// TIA Portal V16 export
// export: Created 2021-11-12T13:31:16.4325674Z, ExportSetting WithDefaults, DisplayName Totally Integrated Automation Portal, DisplayVersion V16 Update 3, DisplayName TIA Portal Version Control Interface, DisplayVersion V16 Update 2, DisplayName TIA Portal Openness, DisplayVersion V16 Update 3, DisplayName SINAMICS Startdrive Advanced, DisplayVersion V16 Update 5, DisplayName SINAMICS Startdrive G130, G150, S120, S150, SINAMICS MV, S210, DisplayVersion V16 Update 5, DisplayName SINAMICS Startdrive G110M, G120, G120C, G120D, G120P, G115D, DisplayVersion V16 Update 5, DisplayName STEP 7 Professional, DisplayVersion V16 Update 3, DisplayName STEP 7 Safety, DisplayVersion V16, DisplayName WinCC UA Professional, DisplayVersion V16 Update 3
FUNCTION_BLOCK "STD_DriveRobotABB"   // FB1226, LAD
TITLE = STD_DriveRobotABB
{ S7_Optimized_Access := 'TRUE' }
VERSION : 0.1
// Logic for robot controller - common for up to 4 robots
// stored: AutoNumber false, IsIECCheckEnabled false, IsRetainMemResEnabled false, MemoryReserve 100, SetENOAutomatically false, UDAEnableTagReadback false
   VAR_INPUT
      IS_ZoneM { ExternalAccessible := 'False'; ExternalVisible := 'False'; ExternalWritable := 'False'} : "UDT_Status_main";   // Main structure from station
      IS_ZoneS { ExternalAccessible := 'False'; ExternalVisible := 'False'; ExternalWritable := 'False'} : "UDT_Zone_Status_specific";   // Specific structure from station
      IS_CtrlSfty : "UDT_DriveRobotABB_ControllerSftyDI";   // Controller safety signals
      IS_CtrlSig : "UDT_DriveRobotABB_ControllerDI";   // Controller non-safety signals
      IB1AckSfty : Bool;   // Reset safety circuit
      IB1En : Bool;   // Enable robots operation / Zone ready to operate
      IB1Init : Bool;   // Initialize robots - start at main
      IB1StartExt : Bool;   // Start robots task - external signal
      IB1StopExt : Bool;   // Stop robots task - external signal
      IB1LimSpd : Bool;   // Set robots maximal speed to safe speed (250mm/s default)
      IB1ReqPause : Bool;   // Request to pause robots jobs
      IB1AlmSupp : Bool;   // Suppress alarms
      IB1Robot1Initialized : Bool := false;   // Robot initialization finished (set 1 if not used)
      IB1Robot2Initialized : Bool := false;   // Robot initialization finished (set 1 if not used)
      IB1Robot3Initialized : Bool := false;   // Robot initialization finished (set 1 if not used)
      IB1Robot4Initialized : Bool := false;   // Robot initialization finished (set 1 if not used)
      IT_CommTmr : Time := T#1000ms;   // Communication timeout
      IT_AckPulseTime : Time := T#200ms;   // Acknowledge pulse length
   END_VAR
   VAR_OUTPUT
      OS_Status : Struct   // Output status
         Main : "UDT_Status_main";
         Specific : "UDT_DriveRobotABB_Status_specific";
         Error : "UDT_Error01";
      END_STRUCT;
      OS_CtrlSig : "UDT_DriveRobotABB_ControllerDO";   // Output signals to controller
      OB1CtrlRun : Bool;   // Controller running in auto mode
      OB1CycleAutostop : Bool;   // Cycle signal Autostop
   END_VAR
   VAR_IN_OUT
      XS_Parameter : "UDT_DriveRobotABB_Parameter";   // Individual parameter structure
      XS_Command : "UDT_DriveRobotABB_Command";   // Individual command structure
   END_VAR
   VAR
      SS_Alarm : Struct   // Device alarms
         CommErr : Bool;   // Communication to robot lost
         EmgStop : Bool;   // Controller emergency stop
         SftyCrct : Bool;   // Controller safety circuit
         NotInAut : Bool;   // Controller is not turned into auto mode
         Res_0_4 : Bool;   // Reserve
         Res_0_5 : Bool;   // Reserve
         Res_0_6 : Bool;   // Reserve
         Res_0_7 : Bool;   // Reserve
      END_STRUCT;
      SS_Warning : Struct   // Device warnings
         SpdRdce : Bool;   // Task speed on touch panel is not 100%
         SimIO : Bool;   // At least one signal is simulated
         SMBBatt : Bool;   // SMB battery charge low
         Temp : Bool;   // CPU temperature higher than 95°C
         NoCycle : Bool;   // None robot is executing task
         Res_0_5 : Bool;   // Reserve
         Res_0_6 : Bool;   // Reserve
         Res_0_7 : Bool;   // Reserve
      END_STRUCT;
      SS_CtrlIn { S7_SetPoint := 'True'} : "UDT_DriveRobotABB_ControllerDI";   // Controller outputs
      SS_CtrlOut { S7_SetPoint := 'True'} : "UDT_DriveRobotABB_ControllerDO";   // Controller inputs
      SB1CollErr : Bool;   // Collective error from device
      SB1CollWrn : Bool;   // Collective warning from device
      SB1CtrlRdy : Bool;   // Controller ready to operation
      SB1ReqInit : Bool;   // Robots init request
      SB1ReqStart : Bool;   // Robots start request
      SB1ReqStartAtMain : Bool;   // Robots start at main request
      SB1InitPE : Bool;   // Robot init request trigger
      SB1StartAtMainPE : Bool;   // Robot init request trigger
      SB1StartExtPE : Bool;   // External start request trigger
      SB1StartTimeOut : Bool;
      ST_CommTmr { S7_SetPoint := 'True'} : TON_TIME;
      ST_RstSfty_TP { S7_SetPoint := 'True'} : TP_TIME;
      ST_RstErr_TP { S7_SetPoint := 'True'} : TP_TIME;
      ST_RstErr_TOF { S7_SetPoint := 'True'} : TOF_TIME;
      ST_ReqStartTimeOut { S7_SetPoint := 'True'} : TON_TIME;
      SS_InitSeqNr : Byte;   // Sequence Initialization
      IEC_Timer_0_Instance { S7_SetPoint := 'True'} : TON_TIME;
      ST_CycleAutostop { S7_SetPoint := 'True'} : TON_TIME;
   END_VAR
   VAR_TEMP
      TS_Status : Struct
         Main : "UDT_Status_main";
         Specific : "UDT_DriveRobotABB_Status_specific";
         Error : "UDT_Error01";
      END_STRUCT;
      TS_Parameter : "UDT_DriveRobotABB_Parameter";
      TS_Command : "UDT_DriveRobotABB_Command";
      TB1CtrlMainCond : Bool;
      TB1AckPulse : Bool;
      TB1AlmSupp : Bool;
      TB1CycleAutostop : Bool;   // Cycle signal Autostop
   END_VAR
   VAR_TEMP   // added for the SCL form of the ladder/FBD networks
      _w1 : Bool;
   END_VAR
BEGIN

REGION Network 1: Clear temporary TS_Status - Main, Specific
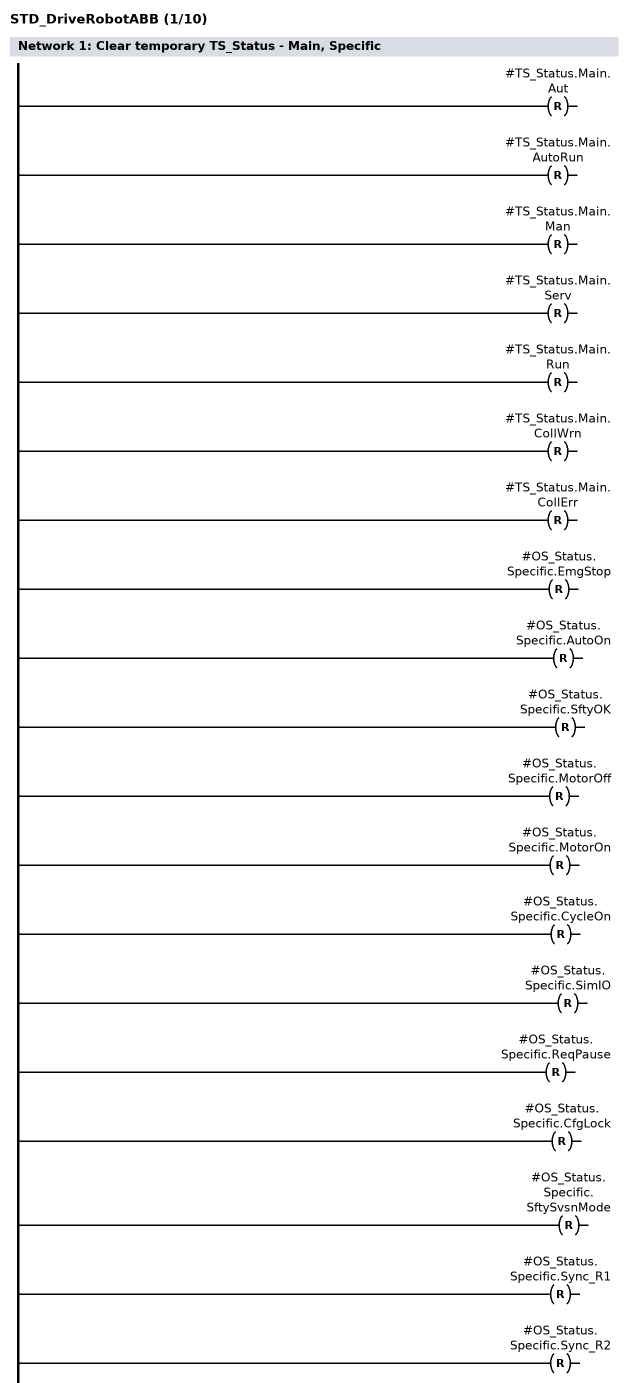
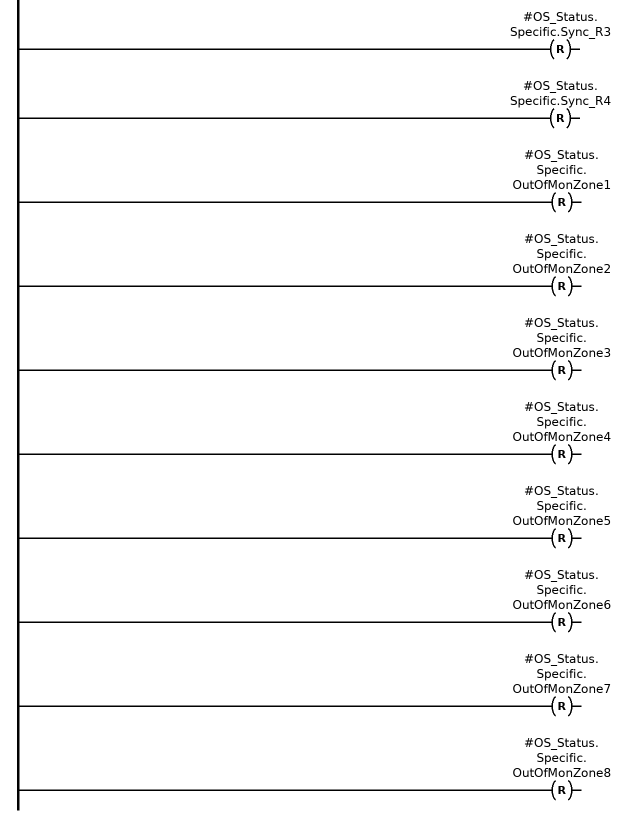
   RUNG wire#powerrail
      R_Coil( #TS_Status.Main.Aut )
   END_RUNG
   RUNG wire#powerrail
      R_Coil( #TS_Status.Main.AutoRun )
   END_RUNG
   RUNG wire#powerrail
      R_Coil( #TS_Status.Main.Man )
   END_RUNG
   RUNG wire#powerrail
      R_Coil( #TS_Status.Main.Serv )
   END_RUNG
   RUNG wire#powerrail
      R_Coil( #TS_Status.Main.Run )
   END_RUNG
   RUNG wire#powerrail
      R_Coil( #TS_Status.Main.CollWrn )
   END_RUNG
   RUNG wire#powerrail
      R_Coil( #TS_Status.Main.CollErr )
   END_RUNG
   RUNG wire#powerrail
      R_Coil( #OS_Status.Specific.EmgStop )
   END_RUNG
   RUNG wire#powerrail
      R_Coil( #OS_Status.Specific.AutoOn )
   END_RUNG
   RUNG wire#powerrail
      R_Coil( #OS_Status.Specific.SftyOK )
   END_RUNG
   RUNG wire#powerrail
      R_Coil( #OS_Status.Specific.MotorOff )
   END_RUNG
   RUNG wire#powerrail
      R_Coil( #OS_Status.Specific.MotorOn )
   END_RUNG
   RUNG wire#powerrail
      R_Coil( #OS_Status.Specific.CycleOn )
   END_RUNG
   RUNG wire#powerrail
      R_Coil( #OS_Status.Specific.SimIO )
   END_RUNG
   RUNG wire#powerrail
      R_Coil( #OS_Status.Specific.ReqPause )
   END_RUNG
   RUNG wire#powerrail
      R_Coil( #OS_Status.Specific.CfgLock )
   END_RUNG
   RUNG wire#powerrail
      R_Coil( #OS_Status.Specific.SftySvsnMode )
   END_RUNG
   RUNG wire#powerrail
      R_Coil( #OS_Status.Specific.Sync_R1 )
   END_RUNG
   RUNG wire#powerrail
      R_Coil( #OS_Status.Specific.Sync_R2 )
   END_RUNG
   RUNG wire#powerrail
      R_Coil( #OS_Status.Specific.Sync_R3 )
   END_RUNG
   RUNG wire#powerrail
      R_Coil( #OS_Status.Specific.Sync_R4 )
   END_RUNG
   RUNG wire#powerrail
      R_Coil( #OS_Status.Specific.OutOfMonZone1 )
   END_RUNG
   RUNG wire#powerrail
      R_Coil( #OS_Status.Specific.OutOfMonZone2 )
   END_RUNG
   RUNG wire#powerrail
      R_Coil( #OS_Status.Specific.OutOfMonZone3 )
   END_RUNG
   RUNG wire#powerrail
      R_Coil( #OS_Status.Specific.OutOfMonZone4 )
   END_RUNG
   RUNG wire#powerrail
      R_Coil( #OS_Status.Specific.OutOfMonZone5 )
   END_RUNG
   RUNG wire#powerrail
      R_Coil( #OS_Status.Specific.OutOfMonZone6 )
   END_RUNG
   RUNG wire#powerrail
      R_Coil( #OS_Status.Specific.OutOfMonZone7 )
   END_RUNG
   RUNG wire#powerrail
      R_Coil( #OS_Status.Specific.OutOfMonZone8 )
   END_RUNG
   // the same network as SCL:
   #TS_Status.Main.Aut := FALSE;
   #TS_Status.Main.AutoRun := FALSE;
   #TS_Status.Main.Man := FALSE;
   #TS_Status.Main.Serv := FALSE;
   #TS_Status.Main.Run := FALSE;
   #TS_Status.Main.CollWrn := FALSE;
   #TS_Status.Main.CollErr := FALSE;
   #OS_Status.Specific.EmgStop := FALSE;
   #OS_Status.Specific.AutoOn := FALSE;
   #OS_Status.Specific.SftyOK := FALSE;
   #OS_Status.Specific.MotorOff := FALSE;
   #OS_Status.Specific.MotorOn := FALSE;
   #OS_Status.Specific.CycleOn := FALSE;
   #OS_Status.Specific.SimIO := FALSE;
   #OS_Status.Specific.ReqPause := FALSE;
   #OS_Status.Specific.CfgLock := FALSE;
   #OS_Status.Specific.SftySvsnMode := FALSE;
   #OS_Status.Specific.Sync_R1 := FALSE;
   #OS_Status.Specific.Sync_R2 := FALSE;
   #OS_Status.Specific.Sync_R3 := FALSE;
   #OS_Status.Specific.Sync_R4 := FALSE;
   #OS_Status.Specific.OutOfMonZone1 := FALSE;
   #OS_Status.Specific.OutOfMonZone2 := FALSE;
   #OS_Status.Specific.OutOfMonZone3 := FALSE;
   #OS_Status.Specific.OutOfMonZone4 := FALSE;
   #OS_Status.Specific.OutOfMonZone5 := FALSE;
   #OS_Status.Specific.OutOfMonZone6 := FALSE;
   #OS_Status.Specific.OutOfMonZone7 := FALSE;
   #OS_Status.Specific.OutOfMonZone8 := FALSE;
END_REGION

REGION Network 2: Copy In/Out variables to temporary variables
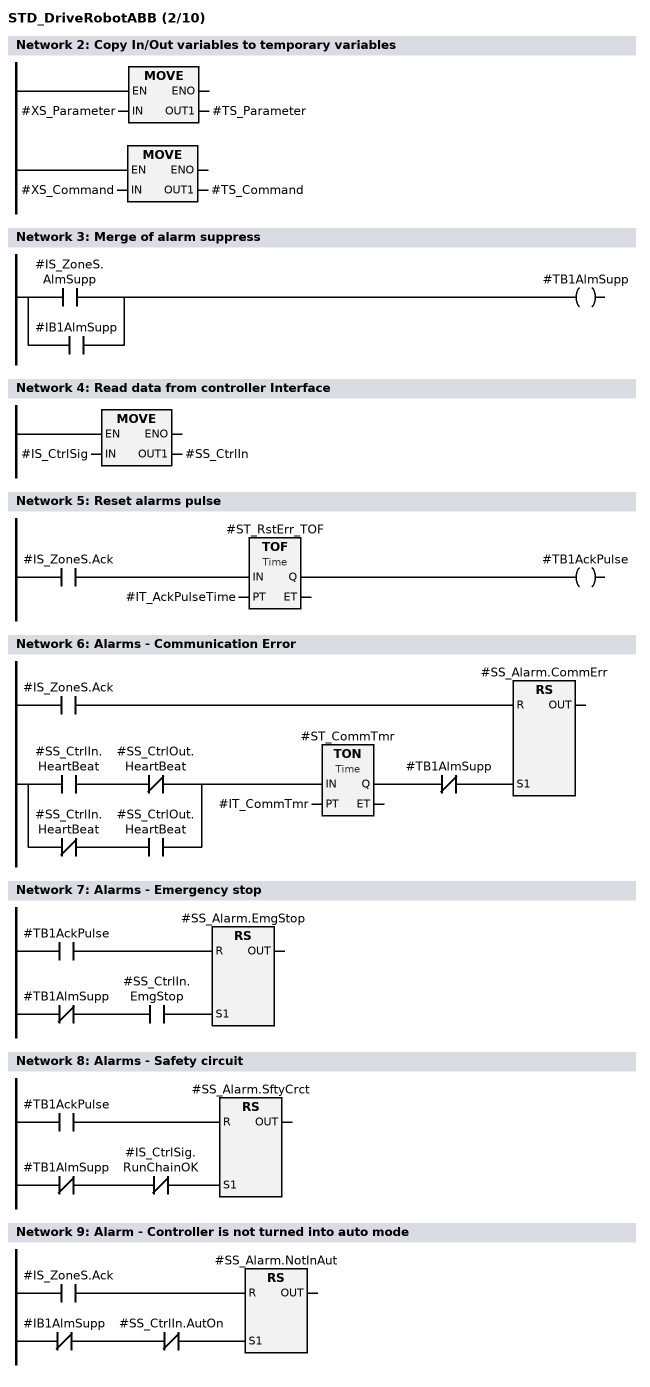
   RUNG wire#powerrail
      { S7_GenerateENO := "TRUE" } Move(in := #XS_Parameter, out1 => #TS_Parameter)
   END_RUNG
   RUNG wire#powerrail
      { S7_GenerateENO := "TRUE" } Move(in := #XS_Command, out1 => #TS_Command)
   END_RUNG
   // the same network as SCL:
   #TS_Parameter := #XS_Parameter;
   #TS_Command := #XS_Command;
END_REGION

REGION Network 3: Merge of alarm suppress
   RUNG wire#powerrail
      Contact( #IS_ZoneS.AlmSupp )
      wire#w1
      Coil( #TB1AlmSupp )
   END_RUNG
   RUNG wire#powerrail
      Contact( #IB1AlmSupp )
   END_RUNG wire#w1
   // the same network as SCL:
   #TB1AlmSupp := #IS_ZoneS.AlmSupp OR #IB1AlmSupp;
END_REGION

REGION Network 4: Read data from controller Interface
   RUNG wire#powerrail
      { S7_GenerateENO := "TRUE" } Move(in := #IS_CtrlSig, out1 => #SS_CtrlIn)
   END_RUNG
   // the same network as SCL:
   #SS_CtrlIn := #IS_CtrlSig;
END_REGION

REGION Network 5: Reset alarms pulse
   RUNG wire#powerrail
      Contact( #IS_ZoneS.Ack )
      { S7_Templates := "time_type := Time" } #ST_RstErr_TOF.TOF(pt := #IT_AckPulseTime, et =>)
      Coil( #TB1AckPulse )
   END_RUNG
   // the same network as SCL:
   #ST_RstErr_TOF(IN := #IS_ZoneS.Ack, PT := #IT_AckPulseTime);   // TOF
   #TB1AckPulse := #ST_RstErr_TOF.Q;
END_REGION

REGION Network 6: Alarms - Communication Error
   RUNG wire#powerrail
      Contact( #IS_ZoneS.Ack )
      S_RS(operand := #SS_Alarm.CommErr, s1 := wire#w2)
   END_RUNG
   RUNG wire#powerrail
      Contact( #SS_CtrlIn.HeartBeat )
      I_Contact( #SS_CtrlOut.HeartBeat )
      wire#w1
      { S7_Templates := "time_type := Time" } #ST_CommTmr.TON(pt := #IT_CommTmr, et =>)
      I_Contact( #TB1AlmSupp )
   END_RUNG wire#w2
   RUNG wire#powerrail
      I_Contact( #SS_CtrlIn.HeartBeat )
      Contact( #SS_CtrlOut.HeartBeat )
   END_RUNG wire#w1
   // the same network as SCL:
   #ST_CommTmr(IN := (#SS_CtrlIn.HeartBeat AND NOT #SS_CtrlOut.HeartBeat) OR (NOT #SS_CtrlIn.HeartBeat AND #SS_CtrlOut.HeartBeat),   // TON
               PT := #IT_CommTmr);
   IF #IS_ZoneS.Ack THEN
       #SS_Alarm.CommErr := FALSE;   // RS flip-flop
   END_IF;
   IF #ST_CommTmr.Q AND NOT #TB1AlmSupp THEN #SS_Alarm.CommErr := TRUE; END_IF;
END_REGION

REGION Network 7: Alarms - Emergency stop
   RUNG wire#powerrail
      Contact( #TB1AckPulse )
      S_RS(operand := #SS_Alarm.EmgStop, s1 := wire#w1)
   END_RUNG
   RUNG wire#powerrail
      I_Contact( #TB1AlmSupp )
      Contact( #SS_CtrlIn.EmgStop )
   END_RUNG wire#w1
   // the same network as SCL:
   IF #TB1AckPulse THEN
       #SS_Alarm.EmgStop := FALSE;   // RS flip-flop
   END_IF;
   IF NOT #TB1AlmSupp AND #SS_CtrlIn.EmgStop THEN #SS_Alarm.EmgStop := TRUE; END_IF;
END_REGION

REGION Network 8: Alarms - Safety circuit
   RUNG wire#powerrail
      Contact( #TB1AckPulse )
      S_RS(operand := #SS_Alarm.SftyCrct, s1 := wire#w1)
   END_RUNG
   RUNG wire#powerrail
      I_Contact( #TB1AlmSupp )
      I_Contact( #IS_CtrlSig.RunChainOK )
   END_RUNG wire#w1
   // the same network as SCL:
   IF #TB1AckPulse THEN
       #SS_Alarm.SftyCrct := FALSE;   // RS flip-flop
   END_IF;
   IF NOT #TB1AlmSupp AND NOT #IS_CtrlSig.RunChainOK THEN #SS_Alarm.SftyCrct := TRUE; END_IF;
END_REGION

REGION Network 9: Alarm - Controller is not turned into auto mode
   RUNG wire#powerrail
      Contact( #IS_ZoneS.Ack )
      S_RS(operand := #SS_Alarm.NotInAut, s1 := wire#w1)
   END_RUNG
   RUNG wire#powerrail
      I_Contact( #IB1AlmSupp )
      I_Contact( #SS_CtrlIn.AutOn )
   END_RUNG wire#w1
   // the same network as SCL:
   IF #IS_ZoneS.Ack THEN
       #SS_Alarm.NotInAut := FALSE;   // RS flip-flop
   END_IF;
   IF NOT #IB1AlmSupp AND NOT #SS_CtrlIn.AutOn THEN #SS_Alarm.NotInAut := TRUE; END_IF;
END_REGION

REGION Network 10: Warning - Simulated IO
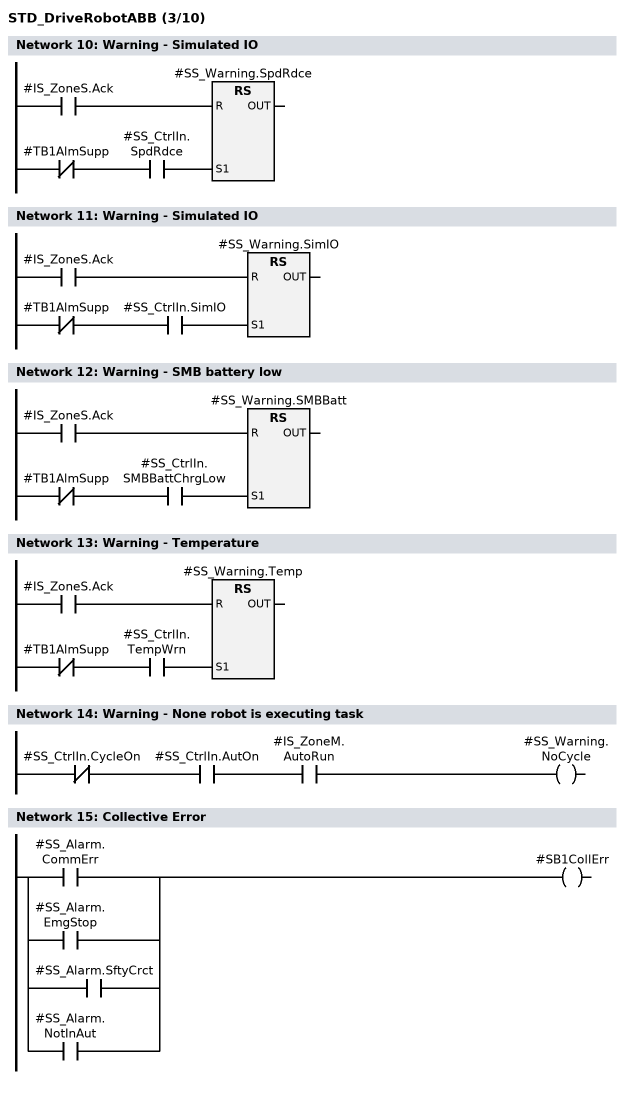
   RUNG wire#powerrail
      Contact( #IS_ZoneS.Ack )
      S_RS(operand := #SS_Warning.SpdRdce, s1 := wire#w1)
   END_RUNG
   RUNG wire#powerrail
      I_Contact( #TB1AlmSupp )
      Contact( #SS_CtrlIn.SpdRdce )
   END_RUNG wire#w1
   // the same network as SCL:
   IF #IS_ZoneS.Ack THEN
       #SS_Warning.SpdRdce := FALSE;   // RS flip-flop
   END_IF;
   IF NOT #TB1AlmSupp AND #SS_CtrlIn.SpdRdce THEN #SS_Warning.SpdRdce := TRUE; END_IF;
END_REGION

REGION Network 11: Warning - Simulated IO
   RUNG wire#powerrail
      Contact( #IS_ZoneS.Ack )
      S_RS(operand := #SS_Warning.SimIO, s1 := wire#w1)
   END_RUNG
   RUNG wire#powerrail
      I_Contact( #TB1AlmSupp )
      Contact( #SS_CtrlIn.SimIO )
   END_RUNG wire#w1
   // the same network as SCL:
   IF #IS_ZoneS.Ack THEN
       #SS_Warning.SimIO := FALSE;   // RS flip-flop
   END_IF;
   IF NOT #TB1AlmSupp AND #SS_CtrlIn.SimIO THEN #SS_Warning.SimIO := TRUE; END_IF;
END_REGION

REGION Network 12: Warning - SMB battery low
   RUNG wire#powerrail
      Contact( #IS_ZoneS.Ack )
      S_RS(operand := #SS_Warning.SMBBatt, s1 := wire#w1)
   END_RUNG
   RUNG wire#powerrail
      I_Contact( #TB1AlmSupp )
      Contact( #SS_CtrlIn.SMBBattChrgLow )
   END_RUNG wire#w1
   // the same network as SCL:
   IF #IS_ZoneS.Ack THEN
       #SS_Warning.SMBBatt := FALSE;   // RS flip-flop
   END_IF;
   IF NOT #TB1AlmSupp AND #SS_CtrlIn.SMBBattChrgLow THEN #SS_Warning.SMBBatt := TRUE; END_IF;
END_REGION

REGION Network 13: Warning - Temperature
   RUNG wire#powerrail
      Contact( #IS_ZoneS.Ack )
      S_RS(operand := #SS_Warning.Temp, s1 := wire#w1)
   END_RUNG
   RUNG wire#powerrail
      I_Contact( #TB1AlmSupp )
      Contact( #SS_CtrlIn.TempWrn )
   END_RUNG wire#w1
   // the same network as SCL:
   IF #IS_ZoneS.Ack THEN
       #SS_Warning.Temp := FALSE;   // RS flip-flop
   END_IF;
   IF NOT #TB1AlmSupp AND #SS_CtrlIn.TempWrn THEN #SS_Warning.Temp := TRUE; END_IF;
END_REGION

REGION Network 14: Warning - None robot is executing task
   RUNG wire#powerrail
      I_Contact( #SS_CtrlIn.CycleOn )
      Contact( #SS_CtrlIn.AutOn )
      Contact( #IS_ZoneM.AutoRun )
      Coil( #SS_Warning.NoCycle )
   END_RUNG
   // the same network as SCL:
   #SS_Warning.NoCycle := NOT #SS_CtrlIn.CycleOn AND #SS_CtrlIn.AutOn AND #IS_ZoneM.AutoRun;
END_REGION

REGION Network 15: Collective Error
   RUNG wire#powerrail
      Contact( #SS_Alarm.CommErr )
      wire#w1
      Coil( #SB1CollErr )
   END_RUNG
   RUNG wire#powerrail
      Contact( #SS_Alarm.EmgStop )
   END_RUNG wire#w1
   RUNG wire#powerrail
      Contact( #SS_Alarm.SftyCrct )
   END_RUNG wire#w1
   RUNG wire#powerrail
      Contact( #SS_Alarm.NotInAut )
   END_RUNG wire#w1
   // the same network as SCL:
   #SB1CollErr := #SS_Alarm.CommErr OR #SS_Alarm.EmgStop OR #SS_Alarm.SftyCrct OR #SS_Alarm.NotInAut;
END_REGION

REGION Network 16: Collective Warning
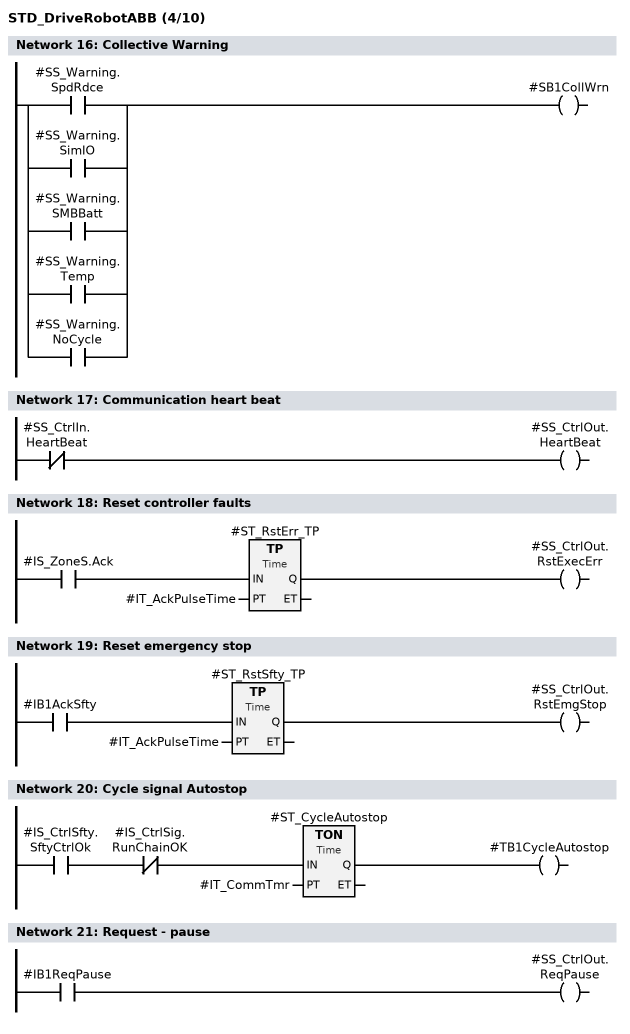
   RUNG wire#powerrail
      Contact( #SS_Warning.SpdRdce )
      wire#w1
      Coil( #SB1CollWrn )
   END_RUNG
   RUNG wire#powerrail
      Contact( #SS_Warning.SimIO )
   END_RUNG wire#w1
   RUNG wire#powerrail
      Contact( #SS_Warning.SMBBatt )
   END_RUNG wire#w1
   RUNG wire#powerrail
      Contact( #SS_Warning.Temp )
   END_RUNG wire#w1
   RUNG wire#powerrail
      Contact( #SS_Warning.NoCycle )
   END_RUNG wire#w1
   // the same network as SCL:
   #SB1CollWrn := #SS_Warning.SpdRdce OR #SS_Warning.SimIO OR #SS_Warning.SMBBatt OR #SS_Warning.Temp OR #SS_Warning.NoCycle;
END_REGION

REGION Network 17: Communication heart beat
   RUNG wire#powerrail
      I_Contact( #SS_CtrlIn.HeartBeat )
      Coil( #SS_CtrlOut.HeartBeat )
   END_RUNG
   // the same network as SCL:
   #SS_CtrlOut.HeartBeat := NOT #SS_CtrlIn.HeartBeat;
END_REGION

REGION Network 18: Reset controller faults
   RUNG wire#powerrail
      Contact( #IS_ZoneS.Ack )
      { S7_Templates := "time_type := Time" } #ST_RstErr_TP.TP(pt := #IT_AckPulseTime, et =>)
      Coil( #SS_CtrlOut.RstExecErr )
   END_RUNG
   // the same network as SCL:
   #ST_RstErr_TP(IN := #IS_ZoneS.Ack, PT := #IT_AckPulseTime);   // TP
   #SS_CtrlOut.RstExecErr := #ST_RstErr_TP.Q;
END_REGION

REGION Network 19: Reset emergency stop
   RUNG wire#powerrail
      Contact( #IB1AckSfty )
      { S7_Templates := "time_type := Time" } #ST_RstSfty_TP.TP(pt := #IT_AckPulseTime, et =>)
      Coil( #SS_CtrlOut.RstEmgStop )
   END_RUNG
   // the same network as SCL:
   #ST_RstSfty_TP(IN := #IB1AckSfty, PT := #IT_AckPulseTime);   // TP
   #SS_CtrlOut.RstEmgStop := #ST_RstSfty_TP.Q;
END_REGION

REGION Network 20: Cycle signal Autostop
   RUNG wire#powerrail
      Contact( #IS_CtrlSfty.SftyCtrlOk )
      I_Contact( #IS_CtrlSig.RunChainOK )
      { S7_Templates := "time_type := Time" } #ST_CycleAutostop.TON(pt := #IT_CommTmr, et =>)
      Coil( #TB1CycleAutostop )
   END_RUNG
   // the same network as SCL:
   #ST_CycleAutostop(IN := #IS_CtrlSfty.SftyCtrlOk AND NOT #IS_CtrlSig.RunChainOK, PT := #IT_CommTmr);   // TON
   #TB1CycleAutostop := #ST_CycleAutostop.Q;
END_REGION

REGION Network 21: Request - pause
   RUNG wire#powerrail
      Contact( #IB1ReqPause )
      Coil( #SS_CtrlOut.ReqPause )
   END_RUNG
   // the same network as SCL:
   #SS_CtrlOut.ReqPause := #IB1ReqPause;
END_REGION

REGION Network 22: Request - Start
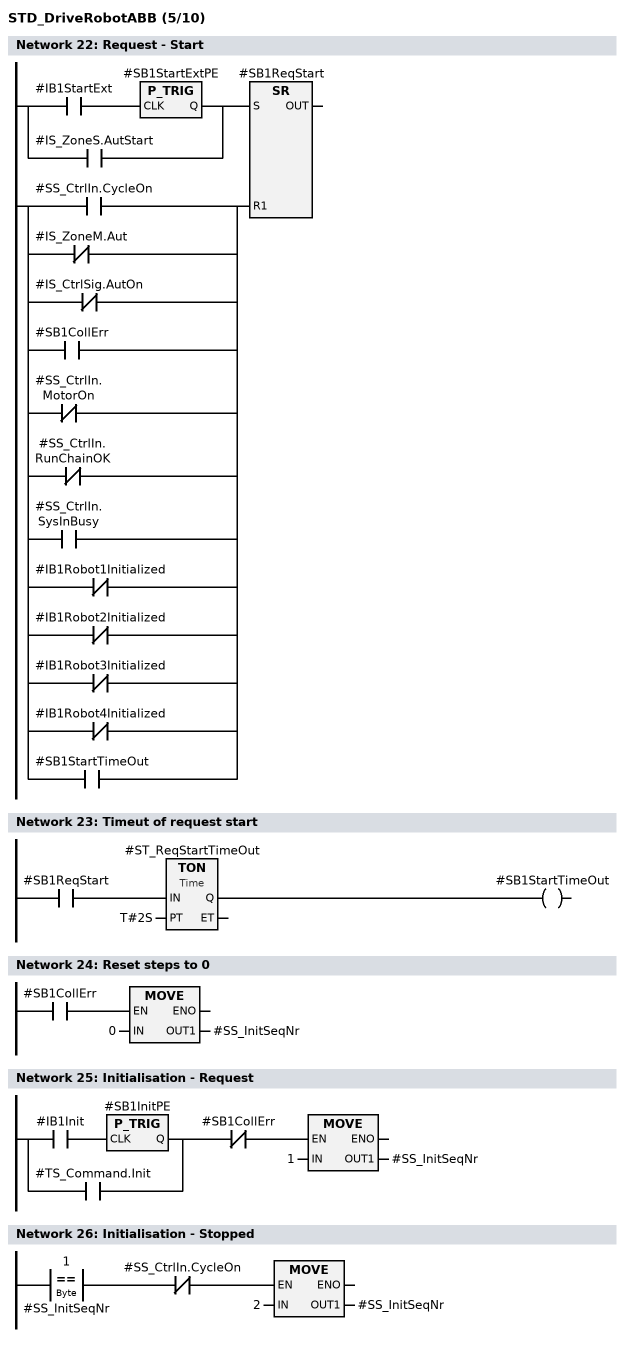
   RUNG wire#powerrail
      Contact( #IB1StartExt )
      P_Trig( #SB1StartExtPE )
      wire#w1
      S_SR(operand := #SB1ReqStart, r1 := wire#w2)
   END_RUNG
   RUNG wire#powerrail
      Contact( #IS_ZoneS.AutStart )
   END_RUNG wire#w1
   RUNG wire#powerrail
      Contact( #SS_CtrlIn.CycleOn )
   END_RUNG wire#w2
   RUNG wire#powerrail
      I_Contact( #IS_ZoneM.Aut )
   END_RUNG wire#w2
   RUNG wire#powerrail
      I_Contact( #IS_CtrlSig.AutOn )
   END_RUNG wire#w2
   RUNG wire#powerrail
      Contact( #SB1CollErr )
   END_RUNG wire#w2
   RUNG wire#powerrail
      I_Contact( #SS_CtrlIn.MotorOn )
   END_RUNG wire#w2
   RUNG wire#powerrail
      I_Contact( #SS_CtrlIn.RunChainOK )
   END_RUNG wire#w2
   RUNG wire#powerrail
      Contact( #SS_CtrlIn.SysInBusy )
   END_RUNG wire#w2
   RUNG wire#powerrail
      I_Contact( #IB1Robot1Initialized )
   END_RUNG wire#w2
   RUNG wire#powerrail
      I_Contact( #IB1Robot2Initialized )
   END_RUNG wire#w2
   RUNG wire#powerrail
      I_Contact( #IB1Robot3Initialized )
   END_RUNG wire#w2
   RUNG wire#powerrail
      I_Contact( #IB1Robot4Initialized )
   END_RUNG wire#w2
   RUNG wire#powerrail
      Contact( #SB1StartTimeOut )
   END_RUNG wire#w2
   // the same network as SCL:
   #_w1 := #IB1StartExt AND NOT #SB1StartExtPE;   // rising edge
   #SB1StartExtPE := #IB1StartExt;
   IF #_w1 OR #IS_ZoneS.AutStart THEN
       #SB1ReqStart := TRUE;   // SR flip-flop
   END_IF;
   IF #SS_CtrlIn.CycleOn OR NOT #IS_ZoneM.Aut OR NOT #IS_CtrlSig.AutOn OR #SB1CollErr OR NOT #SS_CtrlIn.MotorOn OR NOT #SS_CtrlIn.RunChainOK OR #SS_CtrlIn.SysInBusy OR NOT #IB1Robot1Initialized OR NOT #IB1Robot2Initialized OR NOT #IB1Robot3Initialized OR NOT #IB1Robot4Initialized OR #SB1StartTimeOut THEN
       #SB1ReqStart := FALSE;
   END_IF;
END_REGION

REGION Network 23: Timeut of request start
   RUNG wire#powerrail
      Contact( #SB1ReqStart )
      { S7_Templates := "time_type := Time" } #ST_ReqStartTimeOut.TON(pt := T#2S, et =>)
      Coil( #SB1StartTimeOut )
   END_RUNG
   // the same network as SCL:
   #ST_ReqStartTimeOut(IN := #SB1ReqStart, PT := T#2S);   // TON
   #SB1StartTimeOut := #ST_ReqStartTimeOut.Q;
END_REGION

REGION Network 24: Reset steps to 0
   RUNG wire#powerrail
      Contact( #SB1CollErr )
      Move(in := 0, out1 => #SS_InitSeqNr)
   END_RUNG
   // the same network as SCL:
   IF #SB1CollErr THEN #SS_InitSeqNr := 0; END_IF;
END_REGION

REGION Network 25: Initialisation - Request
   RUNG wire#powerrail
      Contact( #IB1Init )
      P_Trig( #SB1InitPE )
      wire#w1
      I_Contact( #SB1CollErr )
      Move(in := 1, out1 => #SS_InitSeqNr)
   END_RUNG
   RUNG wire#powerrail
      Contact( #TS_Command.Init )
   END_RUNG wire#w1
   // the same network as SCL:
   #_w1 := #IB1Init AND NOT #SB1InitPE;   // rising edge
   #SB1InitPE := #IB1Init;
   IF (#_w1 OR #TS_Command.Init) AND NOT #SB1CollErr THEN #SS_InitSeqNr := 1; END_IF;
END_REGION

REGION Network 26: Initialisation - Stopped
   RUNG wire#powerrail
      { S7_Templates := "SrcType := Byte" } EQ_Contact(in1 := 1, in2 := #SS_InitSeqNr)
      I_Contact( #SS_CtrlIn.CycleOn )
      Move(in := 2, out1 => #SS_InitSeqNr)
   END_RUNG
   // the same network as SCL:
   IF (1 = #SS_InitSeqNr) AND NOT #SS_CtrlIn.CycleOn THEN #SS_InitSeqNr := 2; END_IF;
END_REGION

REGION Network 27: Initialization - Started
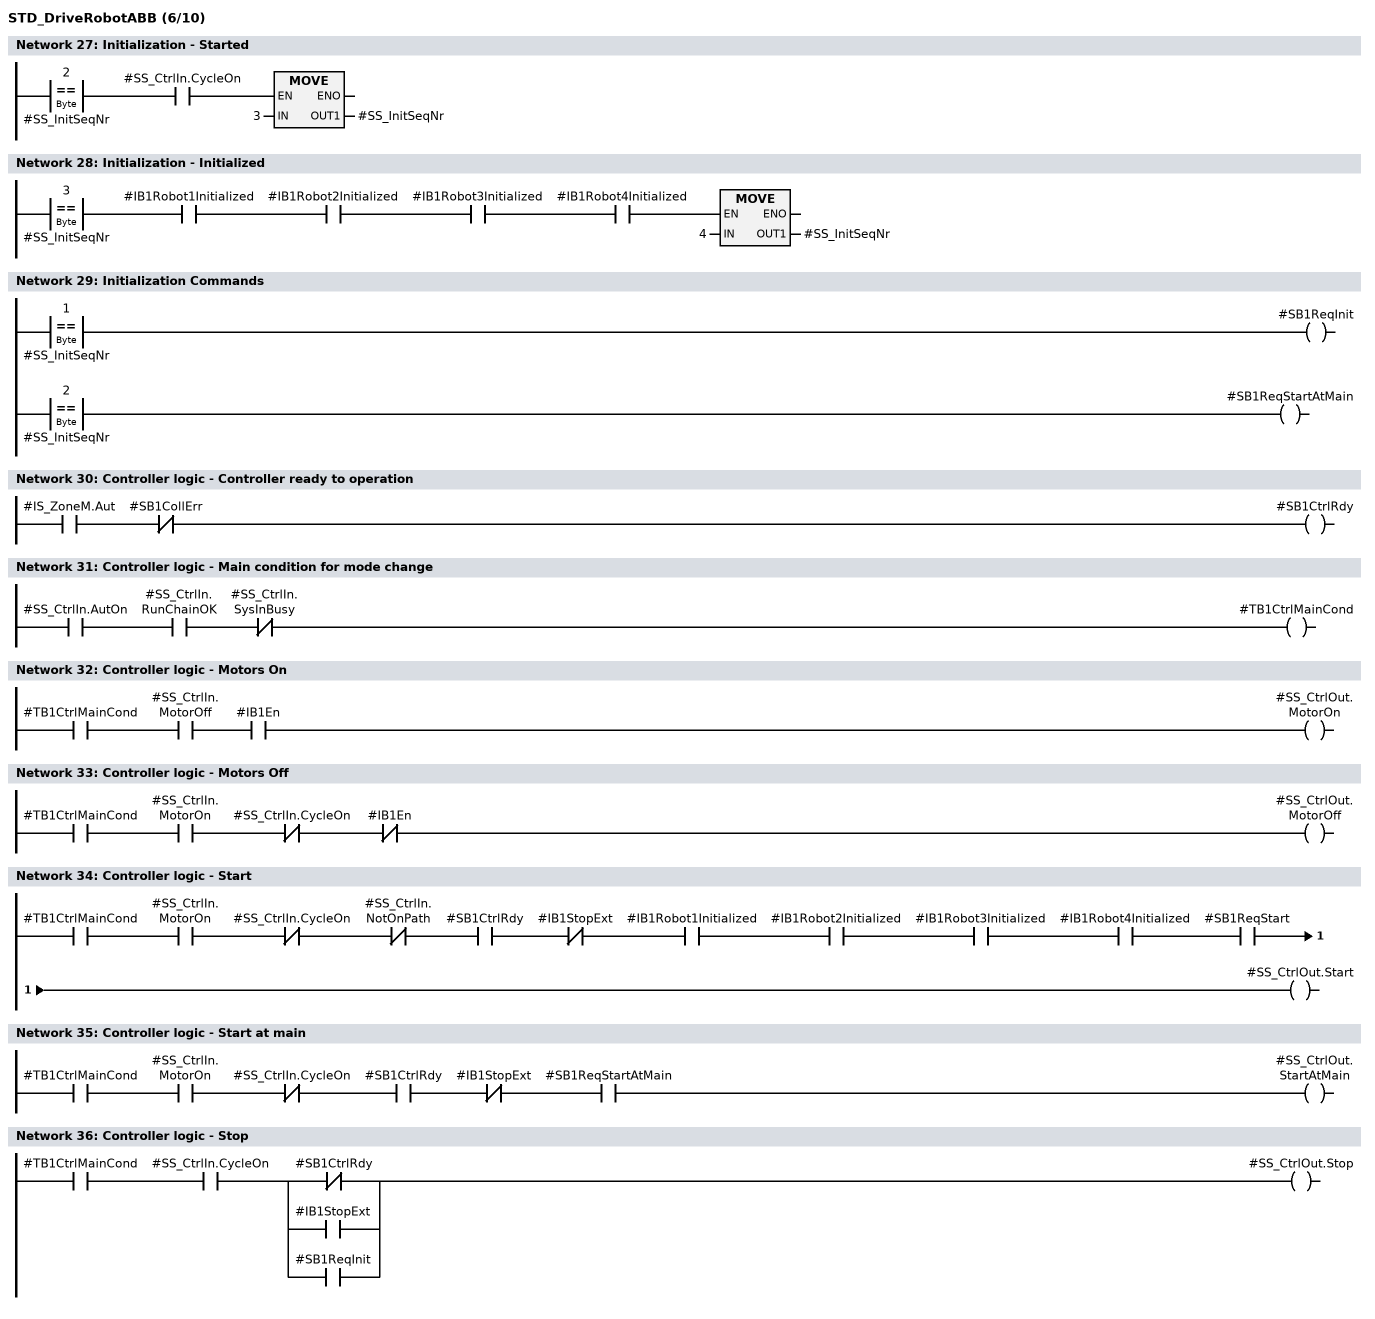
   RUNG wire#powerrail
      { S7_Templates := "SrcType := Byte" } EQ_Contact(in1 := 2, in2 := #SS_InitSeqNr)
      Contact( #SS_CtrlIn.CycleOn )
      Move(in := 3, out1 => #SS_InitSeqNr)
   END_RUNG
   // the same network as SCL:
   IF (2 = #SS_InitSeqNr) AND #SS_CtrlIn.CycleOn THEN #SS_InitSeqNr := 3; END_IF;
END_REGION

REGION Network 28: Initialization - Initialized
   RUNG wire#powerrail
      { S7_Templates := "SrcType := Byte" } EQ_Contact(in1 := 3, in2 := #SS_InitSeqNr)
      Contact( #IB1Robot1Initialized )
      Contact( #IB1Robot2Initialized )
      Contact( #IB1Robot3Initialized )
      Contact( #IB1Robot4Initialized )
      { S7_GenerateENO := "TRUE" } Move(in := 4, out1 => #SS_InitSeqNr)
   END_RUNG
   // the same network as SCL:
   IF (3 = #SS_InitSeqNr) AND #IB1Robot1Initialized AND #IB1Robot2Initialized AND #IB1Robot3Initialized AND #IB1Robot4Initialized THEN
       #SS_InitSeqNr := 4;
   END_IF;
END_REGION

REGION Network 29: Initialization Commands
   RUNG wire#powerrail
      { S7_Templates := "SrcType := Byte" } EQ_Contact(in1 := 1, in2 := #SS_InitSeqNr)
      Coil( #SB1ReqInit )
   END_RUNG
   RUNG wire#powerrail
      { S7_Templates := "SrcType := Byte" } EQ_Contact(in1 := 2, in2 := #SS_InitSeqNr)
      Coil( #SB1ReqStartAtMain )
   END_RUNG
   // the same network as SCL:
   #SB1ReqInit := 1 = #SS_InitSeqNr;
   #SB1ReqStartAtMain := 2 = #SS_InitSeqNr;
END_REGION

REGION Network 30: Controller logic - Controller ready to operation
   RUNG wire#powerrail
      Contact( #IS_ZoneM.Aut )
      I_Contact( #SB1CollErr )
      Coil( #SB1CtrlRdy )
   END_RUNG
   // the same network as SCL:
   #SB1CtrlRdy := #IS_ZoneM.Aut AND NOT #SB1CollErr;
END_REGION

REGION Network 31: Controller logic - Main condition for mode change
   RUNG wire#powerrail
      Contact( #SS_CtrlIn.AutOn )
      Contact( #SS_CtrlIn.RunChainOK )
      I_Contact( #SS_CtrlIn.SysInBusy )
      Coil( #TB1CtrlMainCond )
   END_RUNG
   // the same network as SCL:
   #TB1CtrlMainCond := #SS_CtrlIn.AutOn AND #SS_CtrlIn.RunChainOK AND NOT #SS_CtrlIn.SysInBusy;
END_REGION

REGION Network 32: Controller logic - Motors On
   RUNG wire#powerrail
      Contact( #TB1CtrlMainCond )
      Contact( #SS_CtrlIn.MotorOff )
      Contact( #IB1En )
      Coil( #SS_CtrlOut.MotorOn )
   END_RUNG
   // the same network as SCL:
   #SS_CtrlOut.MotorOn := #TB1CtrlMainCond AND #SS_CtrlIn.MotorOff AND #IB1En;
END_REGION

REGION Network 33: Controller logic - Motors Off
   RUNG wire#powerrail
      Contact( #TB1CtrlMainCond )
      Contact( #SS_CtrlIn.MotorOn )
      I_Contact( #SS_CtrlIn.CycleOn )
      I_Contact( #IB1En )
      Coil( #SS_CtrlOut.MotorOff )
   END_RUNG
   // the same network as SCL:
   #SS_CtrlOut.MotorOff := #TB1CtrlMainCond AND #SS_CtrlIn.MotorOn AND NOT #SS_CtrlIn.CycleOn AND NOT #IB1En;
END_REGION

REGION Network 34: Controller logic - Start
   RUNG wire#powerrail
      Contact( #TB1CtrlMainCond )
      Contact( #SS_CtrlIn.MotorOn )
      I_Contact( #SS_CtrlIn.CycleOn )
      I_Contact( #SS_CtrlIn.NotOnPath )
      Contact( #SB1CtrlRdy )
      I_Contact( #IB1StopExt )
      Contact( #IB1Robot1Initialized )
      Contact( #IB1Robot2Initialized )
      Contact( #IB1Robot3Initialized )
      Contact( #IB1Robot4Initialized )
      Contact( #SB1ReqStart )
      Coil( #SS_CtrlOut.Start )
   END_RUNG
   // the same network as SCL:
   #SS_CtrlOut.Start := #TB1CtrlMainCond AND #SS_CtrlIn.MotorOn AND NOT #SS_CtrlIn.CycleOn AND NOT #SS_CtrlIn.NotOnPath AND #SB1CtrlRdy AND NOT #IB1StopExt AND #IB1Robot1Initialized AND #IB1Robot2Initialized AND #IB1Robot3Initialized AND #IB1Robot4Initialized AND #SB1ReqStart;
END_REGION

REGION Network 35: Controller logic - Start at main
   RUNG wire#powerrail
      Contact( #TB1CtrlMainCond )
      Contact( #SS_CtrlIn.MotorOn )
      I_Contact( #SS_CtrlIn.CycleOn )
      Contact( #SB1CtrlRdy )
      I_Contact( #IB1StopExt )
      Contact( #SB1ReqStartAtMain )
      Coil( #SS_CtrlOut.StartAtMain )
   END_RUNG
   // the same network as SCL:
   #SS_CtrlOut.StartAtMain := #TB1CtrlMainCond AND #SS_CtrlIn.MotorOn AND NOT #SS_CtrlIn.CycleOn AND #SB1CtrlRdy AND NOT #IB1StopExt AND #SB1ReqStartAtMain;
END_REGION

REGION Network 36: Controller logic - Stop
   RUNG wire#powerrail
      Contact( #TB1CtrlMainCond )
      Contact( #SS_CtrlIn.CycleOn )
      wire#w1
      I_Contact( #SB1CtrlRdy )
      wire#w2
      Coil( #SS_CtrlOut.Stop )
   END_RUNG
   RUNG wire#w1
      Contact( #IB1StopExt )
   END_RUNG wire#w2
   RUNG wire#w1
      Contact( #SB1ReqInit )
   END_RUNG wire#w2
   // the same network as SCL:
   #SS_CtrlOut.Stop := #TB1CtrlMainCond AND #SS_CtrlIn.CycleOn AND (NOT #SB1CtrlRdy OR #IB1StopExt OR #SB1ReqInit);
END_REGION

REGION Network 37: Filling the Main status
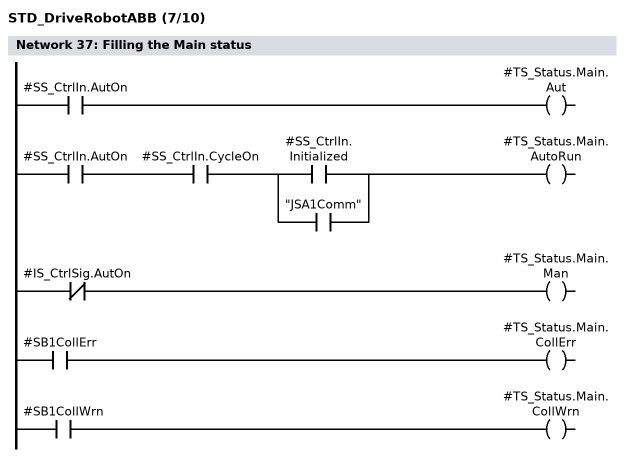
   RUNG wire#powerrail
      Contact( #SS_CtrlIn.AutOn )
      Coil( #TS_Status.Main.Aut )
   END_RUNG
   RUNG wire#powerrail
      Contact( #SS_CtrlIn.AutOn )
      Contact( #SS_CtrlIn.CycleOn )
      wire#w1
      Contact( #SS_CtrlIn.Initialized )
      wire#w2
      Coil( #TS_Status.Main.AutoRun )
   END_RUNG
   RUNG wire#w1
      Contact( "JSA1Comm" )
   END_RUNG wire#w2
   RUNG wire#powerrail
      I_Contact( #IS_CtrlSig.AutOn )
      Coil( #TS_Status.Main.Man )
   END_RUNG
   RUNG wire#powerrail
      Contact( #SB1CollErr )
      Coil( #TS_Status.Main.CollErr )
   END_RUNG
   RUNG wire#powerrail
      Contact( #SB1CollWrn )
      Coil( #TS_Status.Main.CollWrn )
   END_RUNG
   // the same network as SCL:
   #TS_Status.Main.Aut := #SS_CtrlIn.AutOn;
   #TS_Status.Main.AutoRun := #SS_CtrlIn.AutOn AND #SS_CtrlIn.CycleOn AND (#SS_CtrlIn.Initialized OR "JSA1Comm");
   #TS_Status.Main.Man := NOT #IS_CtrlSig.AutOn;
   #TS_Status.Main.CollErr := #SB1CollErr;
   #TS_Status.Main.CollWrn := #SB1CollWrn;
END_REGION

REGION Network 38: Filling the Specific status
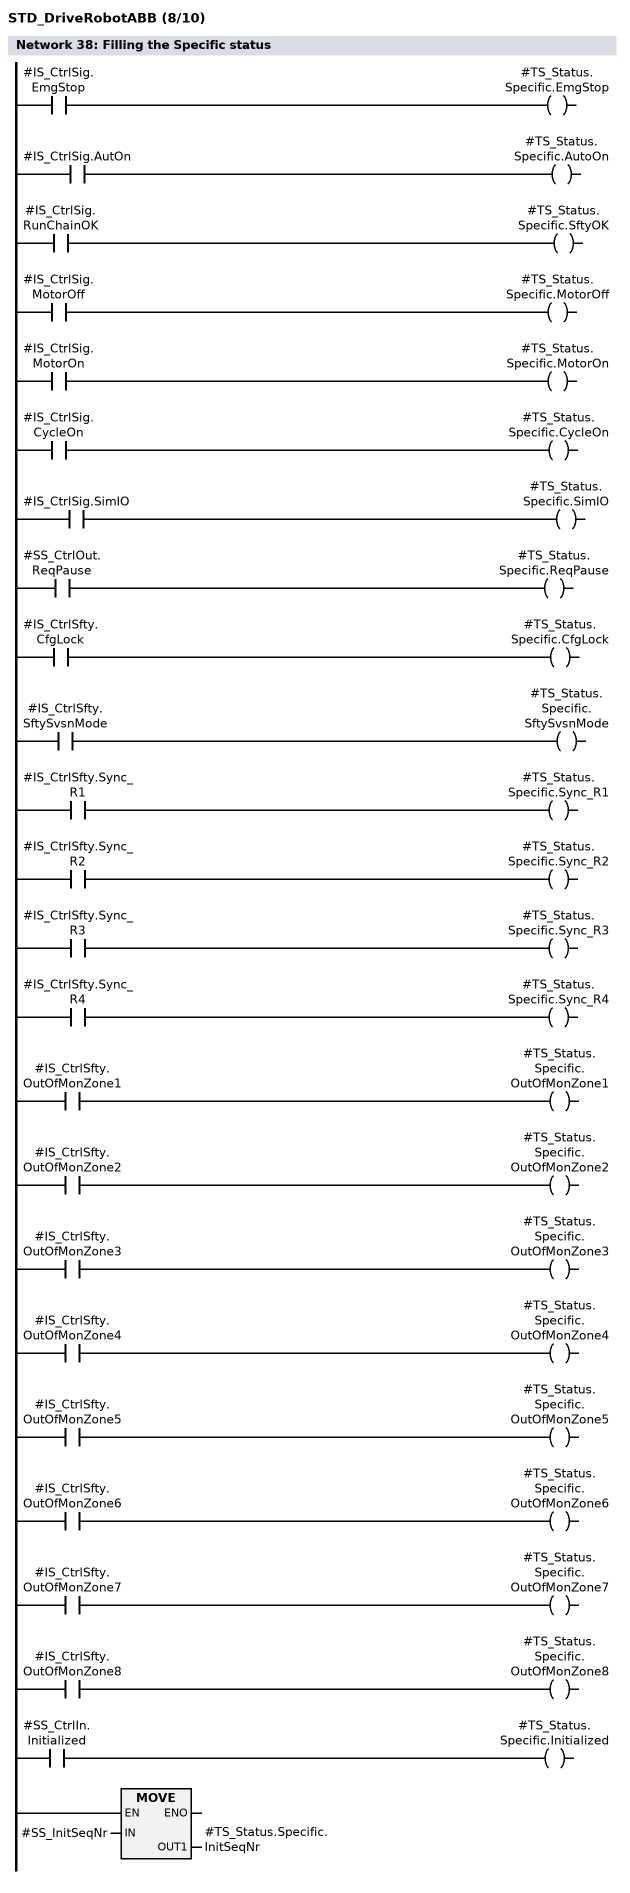
   RUNG wire#powerrail
      Contact( #IS_CtrlSig.EmgStop )
      Coil( #TS_Status.Specific.EmgStop )
   END_RUNG
   RUNG wire#powerrail
      Contact( #IS_CtrlSig.AutOn )
      Coil( #TS_Status.Specific.AutoOn )
   END_RUNG
   RUNG wire#powerrail
      Contact( #IS_CtrlSig.RunChainOK )
      Coil( #TS_Status.Specific.SftyOK )
   END_RUNG
   RUNG wire#powerrail
      Contact( #IS_CtrlSig.MotorOff )
      Coil( #TS_Status.Specific.MotorOff )
   END_RUNG
   RUNG wire#powerrail
      Contact( #IS_CtrlSig.MotorOn )
      Coil( #TS_Status.Specific.MotorOn )
   END_RUNG
   RUNG wire#powerrail
      Contact( #IS_CtrlSig.CycleOn )
      Coil( #TS_Status.Specific.CycleOn )
   END_RUNG
   RUNG wire#powerrail
      Contact( #IS_CtrlSig.SimIO )
      Coil( #TS_Status.Specific.SimIO )
   END_RUNG
   RUNG wire#powerrail
      Contact( #SS_CtrlOut.ReqPause )
      Coil( #TS_Status.Specific.ReqPause )
   END_RUNG
   RUNG wire#powerrail
      Contact( #IS_CtrlSfty.CfgLock )
      Coil( #TS_Status.Specific.CfgLock )
   END_RUNG
   RUNG wire#powerrail
      Contact( #IS_CtrlSfty.SftySvsnMode )
      Coil( #TS_Status.Specific.SftySvsnMode )
   END_RUNG
   RUNG wire#powerrail
      Contact( #IS_CtrlSfty.Sync_R1 )
      Coil( #TS_Status.Specific.Sync_R1 )
   END_RUNG
   RUNG wire#powerrail
      Contact( #IS_CtrlSfty.Sync_R2 )
      Coil( #TS_Status.Specific.Sync_R2 )
   END_RUNG
   RUNG wire#powerrail
      Contact( #IS_CtrlSfty.Sync_R3 )
      Coil( #TS_Status.Specific.Sync_R3 )
   END_RUNG
   RUNG wire#powerrail
      Contact( #IS_CtrlSfty.Sync_R4 )
      Coil( #TS_Status.Specific.Sync_R4 )
   END_RUNG
   RUNG wire#powerrail
      Contact( #IS_CtrlSfty.OutOfMonZone1 )
      Coil( #TS_Status.Specific.OutOfMonZone1 )
   END_RUNG
   RUNG wire#powerrail
      Contact( #IS_CtrlSfty.OutOfMonZone2 )
      Coil( #TS_Status.Specific.OutOfMonZone2 )
   END_RUNG
   RUNG wire#powerrail
      Contact( #IS_CtrlSfty.OutOfMonZone3 )
      Coil( #TS_Status.Specific.OutOfMonZone3 )
   END_RUNG
   RUNG wire#powerrail
      Contact( #IS_CtrlSfty.OutOfMonZone4 )
      Coil( #TS_Status.Specific.OutOfMonZone4 )
   END_RUNG
   RUNG wire#powerrail
      Contact( #IS_CtrlSfty.OutOfMonZone5 )
      Coil( #TS_Status.Specific.OutOfMonZone5 )
   END_RUNG
   RUNG wire#powerrail
      Contact( #IS_CtrlSfty.OutOfMonZone6 )
      Coil( #TS_Status.Specific.OutOfMonZone6 )
   END_RUNG
   RUNG wire#powerrail
      Contact( #IS_CtrlSfty.OutOfMonZone7 )
      Coil( #TS_Status.Specific.OutOfMonZone7 )
   END_RUNG
   RUNG wire#powerrail
      Contact( #IS_CtrlSfty.OutOfMonZone8 )
      Coil( #TS_Status.Specific.OutOfMonZone8 )
   END_RUNG
   RUNG wire#powerrail
      Contact( #SS_CtrlIn.Initialized )
      Coil( #TS_Status.Specific.Initialized )
   END_RUNG
   RUNG wire#powerrail
      { S7_GenerateENO := "TRUE" } Move(in := #SS_InitSeqNr, out1 => #TS_Status.Specific.InitSeqNr)
   END_RUNG
   // the same network as SCL:
   #TS_Status.Specific.EmgStop := #IS_CtrlSig.EmgStop;
   #TS_Status.Specific.AutoOn := #IS_CtrlSig.AutOn;
   #TS_Status.Specific.SftyOK := #IS_CtrlSig.RunChainOK;
   #TS_Status.Specific.MotorOff := #IS_CtrlSig.MotorOff;
   #TS_Status.Specific.MotorOn := #IS_CtrlSig.MotorOn;
   #TS_Status.Specific.CycleOn := #IS_CtrlSig.CycleOn;
   #TS_Status.Specific.SimIO := #IS_CtrlSig.SimIO;
   #TS_Status.Specific.ReqPause := #SS_CtrlOut.ReqPause;
   #TS_Status.Specific.CfgLock := #IS_CtrlSfty.CfgLock;
   #TS_Status.Specific.SftySvsnMode := #IS_CtrlSfty.SftySvsnMode;
   #TS_Status.Specific.Sync_R1 := #IS_CtrlSfty.Sync_R1;
   #TS_Status.Specific.Sync_R2 := #IS_CtrlSfty.Sync_R2;
   #TS_Status.Specific.Sync_R3 := #IS_CtrlSfty.Sync_R3;
   #TS_Status.Specific.Sync_R4 := #IS_CtrlSfty.Sync_R4;
   #TS_Status.Specific.OutOfMonZone1 := #IS_CtrlSfty.OutOfMonZone1;
   #TS_Status.Specific.OutOfMonZone2 := #IS_CtrlSfty.OutOfMonZone2;
   #TS_Status.Specific.OutOfMonZone3 := #IS_CtrlSfty.OutOfMonZone3;
   #TS_Status.Specific.OutOfMonZone4 := #IS_CtrlSfty.OutOfMonZone4;
   #TS_Status.Specific.OutOfMonZone5 := #IS_CtrlSfty.OutOfMonZone5;
   #TS_Status.Specific.OutOfMonZone6 := #IS_CtrlSfty.OutOfMonZone6;
   #TS_Status.Specific.OutOfMonZone7 := #IS_CtrlSfty.OutOfMonZone7;
   #TS_Status.Specific.OutOfMonZone8 := #IS_CtrlSfty.OutOfMonZone8;
   #TS_Status.Specific.Initialized := #SS_CtrlIn.Initialized;
   #TS_Status.Specific.InitSeqNr := #SS_InitSeqNr;
END_REGION

REGION Network 39: Reset Commands
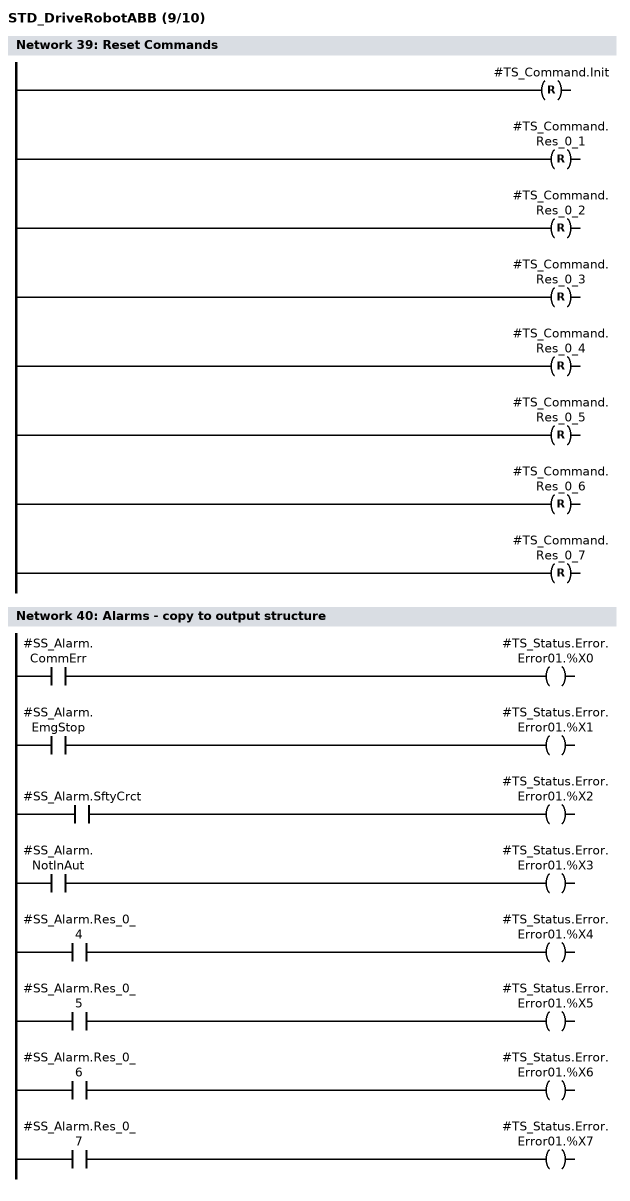
   RUNG wire#powerrail
      R_Coil( #TS_Command.Init )
   END_RUNG
   RUNG wire#powerrail
      R_Coil( #TS_Command.Res_0_1 )
   END_RUNG
   RUNG wire#powerrail
      R_Coil( #TS_Command.Res_0_2 )
   END_RUNG
   RUNG wire#powerrail
      R_Coil( #TS_Command.Res_0_3 )
   END_RUNG
   RUNG wire#powerrail
      R_Coil( #TS_Command.Res_0_4 )
   END_RUNG
   RUNG wire#powerrail
      R_Coil( #TS_Command.Res_0_5 )
   END_RUNG
   RUNG wire#powerrail
      R_Coil( #TS_Command.Res_0_6 )
   END_RUNG
   RUNG wire#powerrail
      R_Coil( #TS_Command.Res_0_7 )
   END_RUNG
   // the same network as SCL:
   #TS_Command.Init := FALSE;
   #TS_Command.Res_0_1 := FALSE;
   #TS_Command.Res_0_2 := FALSE;
   #TS_Command.Res_0_3 := FALSE;
   #TS_Command.Res_0_4 := FALSE;
   #TS_Command.Res_0_5 := FALSE;
   #TS_Command.Res_0_6 := FALSE;
   #TS_Command.Res_0_7 := FALSE;
END_REGION

REGION Network 40: Alarms - copy to output structure
   RUNG wire#powerrail
      Contact( #SS_Alarm.CommErr )
      Coil( #TS_Status.Error.Error01.%X0 )
   END_RUNG
   RUNG wire#powerrail
      Contact( #SS_Alarm.EmgStop )
      Coil( #TS_Status.Error.Error01.%X1 )
   END_RUNG
   RUNG wire#powerrail
      Contact( #SS_Alarm.SftyCrct )
      Coil( #TS_Status.Error.Error01.%X2 )
   END_RUNG
   RUNG wire#powerrail
      Contact( #SS_Alarm.NotInAut )
      Coil( #TS_Status.Error.Error01.%X3 )
   END_RUNG
   RUNG wire#powerrail
      Contact( #SS_Alarm.Res_0_4 )
      Coil( #TS_Status.Error.Error01.%X4 )
   END_RUNG
   RUNG wire#powerrail
      Contact( #SS_Alarm.Res_0_5 )
      Coil( #TS_Status.Error.Error01.%X5 )
   END_RUNG
   RUNG wire#powerrail
      Contact( #SS_Alarm.Res_0_6 )
      Coil( #TS_Status.Error.Error01.%X6 )
   END_RUNG
   RUNG wire#powerrail
      Contact( #SS_Alarm.Res_0_7 )
      Coil( #TS_Status.Error.Error01.%X7 )
   END_RUNG
   // the same network as SCL:
   #TS_Status.Error.Error01.%X0 := #SS_Alarm.CommErr;
   #TS_Status.Error.Error01.%X1 := #SS_Alarm.EmgStop;
   #TS_Status.Error.Error01.%X2 := #SS_Alarm.SftyCrct;
   #TS_Status.Error.Error01.%X3 := #SS_Alarm.NotInAut;
   #TS_Status.Error.Error01.%X4 := #SS_Alarm.Res_0_4;
   #TS_Status.Error.Error01.%X5 := #SS_Alarm.Res_0_5;
   #TS_Status.Error.Error01.%X6 := #SS_Alarm.Res_0_6;
   #TS_Status.Error.Error01.%X7 := #SS_Alarm.Res_0_7;
END_REGION

REGION Network 41: Warnings - copy to output structure
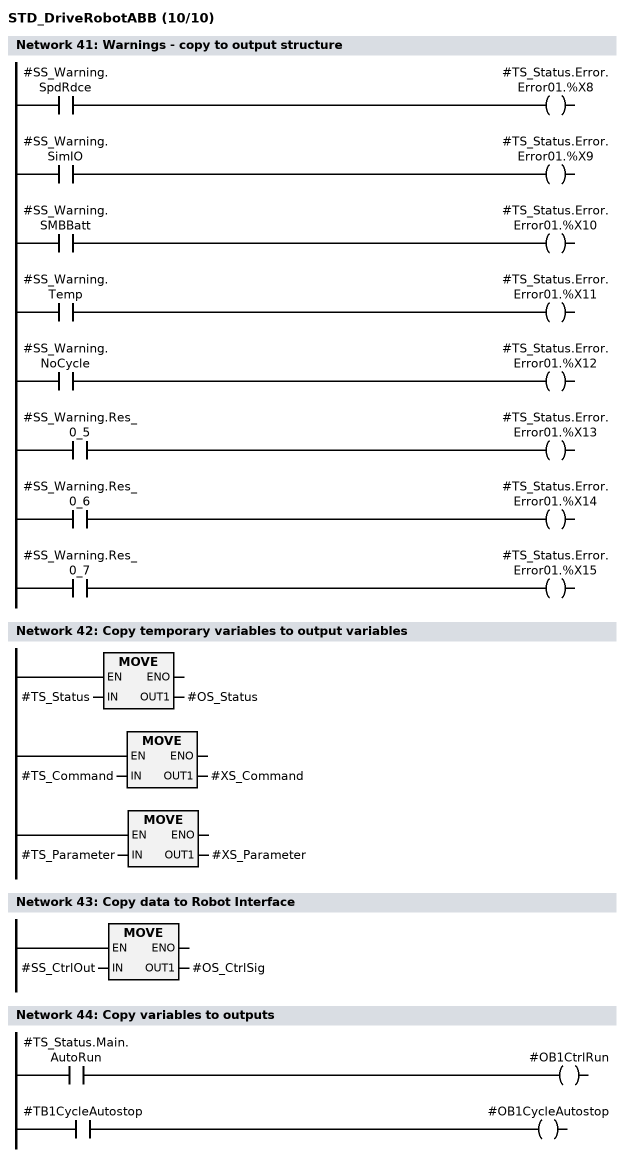
   RUNG wire#powerrail
      Contact( #SS_Warning.SpdRdce )
      Coil( #TS_Status.Error.Error01.%X8 )
   END_RUNG
   RUNG wire#powerrail
      Contact( #SS_Warning.SimIO )
      Coil( #TS_Status.Error.Error01.%X9 )
   END_RUNG
   RUNG wire#powerrail
      Contact( #SS_Warning.SMBBatt )
      Coil( #TS_Status.Error.Error01.%X10 )
   END_RUNG
   RUNG wire#powerrail
      Contact( #SS_Warning.Temp )
      Coil( #TS_Status.Error.Error01.%X11 )
   END_RUNG
   RUNG wire#powerrail
      Contact( #SS_Warning.NoCycle )
      Coil( #TS_Status.Error.Error01.%X12 )
   END_RUNG
   RUNG wire#powerrail
      Contact( #SS_Warning.Res_0_5 )
      Coil( #TS_Status.Error.Error01.%X13 )
   END_RUNG
   RUNG wire#powerrail
      Contact( #SS_Warning.Res_0_6 )
      Coil( #TS_Status.Error.Error01.%X14 )
   END_RUNG
   RUNG wire#powerrail
      Contact( #SS_Warning.Res_0_7 )
      Coil( #TS_Status.Error.Error01.%X15 )
   END_RUNG
   // the same network as SCL:
   #TS_Status.Error.Error01.%X8 := #SS_Warning.SpdRdce;
   #TS_Status.Error.Error01.%X9 := #SS_Warning.SimIO;
   #TS_Status.Error.Error01.%X10 := #SS_Warning.SMBBatt;
   #TS_Status.Error.Error01.%X11 := #SS_Warning.Temp;
   #TS_Status.Error.Error01.%X12 := #SS_Warning.NoCycle;
   #TS_Status.Error.Error01.%X13 := #SS_Warning.Res_0_5;
   #TS_Status.Error.Error01.%X14 := #SS_Warning.Res_0_6;
   #TS_Status.Error.Error01.%X15 := #SS_Warning.Res_0_7;
END_REGION

REGION Network 42: Copy temporary variables to output variables
   RUNG wire#powerrail
      { S7_GenerateENO := "TRUE" } Move(in := #TS_Status, out1 => #OS_Status)
   END_RUNG
   RUNG wire#powerrail
      { S7_GenerateENO := "TRUE" } Move(in := #TS_Command, out1 => #XS_Command)
   END_RUNG
   RUNG wire#powerrail
      { S7_GenerateENO := "TRUE" } Move(in := #TS_Parameter, out1 => #XS_Parameter)
   END_RUNG
   // the same network as SCL:
   #OS_Status := #TS_Status;
   #XS_Command := #TS_Command;
   #XS_Parameter := #TS_Parameter;
END_REGION

REGION Network 43: Copy data to Robot Interface
   RUNG wire#powerrail
      { S7_GenerateENO := "TRUE" } Move(in := #SS_CtrlOut, out1 => #OS_CtrlSig)
   END_RUNG
   // the same network as SCL:
   #OS_CtrlSig := #SS_CtrlOut;
END_REGION

REGION Network 44: Copy variables to outputs
   RUNG wire#powerrail
      Contact( #TS_Status.Main.AutoRun )
      Coil( #OB1CtrlRun )
   END_RUNG
   RUNG wire#powerrail
      Contact( #TB1CycleAutostop )
      Coil( #OB1CycleAutostop )
   END_RUNG
   // the same network as SCL:
   #OB1CtrlRun := #TS_Status.Main.AutoRun;
   #OB1CycleAutostop := #TB1CycleAutostop;
END_REGION
END_FUNCTION_BLOCK
